// TIA Portal V19 export
TYPE "Thickness_Par"
   STRUCT
      SensorON : Bool;
      Trigger_interval : Real;
      NG_Measures_ToFault : Int;   // Number of out-of-range Thickness Measurements Triggering the Alarm
      BypassAutoReset : Int;
      Tolerance_Min : Real;
      Tolerance_Max : Real;
      MES_RecordChange_ThresholdMin : Real;   // Positive Threshold for Communication of Average Thickness Change
      MES_RecordChange_ThresholdMax : Real;   // Negative Threshold for Communication of Average Thickness Change
   END_STRUCT;
END_TYPE
